KUKA KRL data list: DisableRSI_Pos.dat

&ACCESS RV
&REL 1
DEFDAT  DisableRSI_Pos PUBLIC

ENDDAT
